FUNCTION_BLOCK FB_SEW_Movisafe IMPLEMENTS I_SEW_Movisafe
VAR_INPUT
	bSetSTO : BOOL;
END_VAR
VAR_OUTPUT
END_VAR
VAR
END_VAR

PROPERTY bSTO : BOOL
GET
bSTO := bSetSTO;
END_GET
END_PROPERTY

END_FUNCTION_BLOCK

(* stored: Version 1.1.0.1, ProductVersion 3.1.4024.12
   POU FB_SEW_Movisafe: Id {cb41f74c-7b55-0a32-3379-548c117bfa18}, SpecialFunc None
   Property bSTO: Id {97e70496-5f1b-0c90-39a4-9af65fa80751}
   Get Get: Id {b40ef4ad-cfa1-0939-170c-e491bc50d3cc} *)
